// TIA Portal V18 export
// export: Created 2025-12-01T17:52:58.5389529Z, ExportSetting None, DisplayName Totally Integrated Automation Portal, DisplayVersion V18 Update 5, DisplayName TIA Portal Openness, DisplayVersion V18 Update 5, DisplayName TIA Portal Teamcenter Gateway, DisplayVersion V18, DisplayName TIA Portal Version Control Interface, DisplayVersion V18, DisplayName STEP 7 Professional, DisplayVersion V18 Update 5, DisplayName STEP 7 Safety, DisplayVersion V18, DisplayName WinCC Professional, DisplayVersion V18 Update 5
Screen "220_Cylinder_B1"  1280x800, Number=220, Template=02ManualUnit1
  ScreenLayer "Layer_0"
    FaceplateInstance "Cylinder_S71500_TP700_1" at 0,85 size 1279x80  FaceplateTypeName=03 FunctionBlocks@$@101 Cylinder@$@101.2 HMI@$@S7-1500@$@Cylinder_S71500_TP700 V 0.0.29
      Cy := STxxxCylinder005
      CylinderName := Cyl name
      HomeButtonName := Cyl go home button
      WorkButtonName := Cyl go work button
      HomeQaddress := Cyl home Q
      HomeIaddress := Cyl home I
      WorkIaddress := Cyl work I
      WorkQaddress := Cyl work Q
    FaceplateInstance "Cylinder_S71500_TP700_3" at 0,160 size 1279x80  FaceplateTypeName=03 FunctionBlocks@$@101 Cylinder@$@101.2 HMI@$@S7-1500@$@Cylinder_S71500_TP700 V 0.0.29
      Cy := STxxxCylinder006
      CylinderName := Cyl name
      HomeButtonName := Cyl go home button
      WorkButtonName := Cyl go work button
      HomeQaddress := Cyl home Q
      HomeIaddress := Cyl home I
      WorkIaddress := Cyl work I
      WorkQaddress := Cyl work Q
    Button "btnMenu4" at 384,725 size 128x75  TextOff="B-读码器 806A1 / B-CodeReader 806A1", TextOn="B-读码器 806A1 / B-CodeReader 806A1"
      on Click: ActivateScreen(Screen name := 222 Scanner_806A1, Object number := 0)
    Button "btnMenu5" at 512,725 size 128x75  TextOff="B-气缸2 / B-Cylinder2", TextOn="B-气缸2 / B-Cylinder2"
      on Click: ActivateScreen(Screen name := 226_Cylinder_B2, Object number := 0)
    Button "btnMenu6" at 640,725 size 128x75  TextOff="B-压机 375A1 / B-Press 375A1", TextOn="B-压机 375A1 / B-Press 375A1"
      on Click: ActivateScreen(Screen name := 227 Kistler_375A1, Object number := 0)
    Button "btnMenu7" at 896,725 size 128x75
    Button "btnMenu6_1" at 768,725 size 128x75
    Button "btnMenu7_1" at 1024,725 size 128x75
    Button "按钮_9" at 128,725 size 128x75  PictureOff=向右箭头_0, TextOff="B-气缸1 / B-Cylinder1", TextOn="B-气缸1 / B-Cylinder1"
      on Click: ActivateScreen(Screen name := , Object number := 0)
    Button "btnMenu4_1" at 256,725 size 128x75  TextOff="B-压机 372A1 / B-Press 372A1", TextOn="B-压机 372A1 / B-Press 372A1"
      on Click: ActivateScreen(Screen name := 221 Kistler__372A1, Object number := 0)
    GraphicView "图形视图_1" at 201,241 size 455x447  Picture=图形_49
